PROGRAM PRG_TEST
VAR
	fbInductiveSensorTest : FB_Component_InductiveSensor_Test;
END_VAR

TcUnit.RUN();

END_PROGRAM

(* stored: Version 1.1.0.1, ProductVersion 3.1.4024.15
   POU PRG_TEST: Id {21c1260b-e693-4fab-a947-7480831557b1}, SpecialFunc None *)
